(* IEC 61131-3 sources: programs/VI-54/VI-54_20171205/VI-54_20171205/Stations/Screen/LseClass170718/Class/ParameterLogFile, 1 file *)

(* ---- ParameterLogFile.st ---- *)
(*!
<Class
	Name               = "ParameterLogFile"
	Revision           = "0.0"
	RealtimeTask       = "false"
	CyclicTask         = "false"
	BackgroundTask     = "false"
	Sigmatek           = "false"
	OSInterface        = "false"
	HighPriority       = "false"
	Automatic          = "false"
	UpdateMode         = "Prescan"
	SharedCommandTable = "true"
	Objectsize         = "(540,120)">
	<Channels>
	</Channels>
	<Network Name="ParameterLogFile">
		<!-- List of Components in this network -->
		<Components>
			<Object
				Name       = "_base"
				Class      = "_Global"
				Position   = "(218,120)"
				Visualized = "true"
				Remotely   = "true">
				<Channels>
					<Server Name="Server0">
						<OPCSettings WriteProtected="false"/>
					</Server>
					<Client Name="Lse"/>
				</Channels>
			</Object>
		</Components>
		<Comments>
		</Comments>
		<!-- List of Connections in this network -->
		<Connections>
			<Connection Source="this.Server0" Destination="_base.Server0" Vertices="(690,210),(518,210),"/>
			<Connection Source="_base.Lse" Destination="this.Lse" Vertices="(218,210),(38,210),"/>
		</Connections>
		<!-- Headerfiles -->
		<Options>
		</Options>
	</Network>
</Class>
*)
#pragma using _Global

ParameterLogFile : CLASS
: _Global
  //Servers:
  //Clients:
  //Variables:
		VariableInformation 	: ^_EDITOR;
		WindowNbr 	: UDINT;
		ActualValue 	: DINT;
		ActualMin 	: DINT;
		ActualMax 	: DINT;
  //Functions:
				//! <Function Comment="method is called right before the kernel wants to open a toucheditor&#13;&#10;the parameter &apos;pe&apos; is a pointer to structure where the whole editorinformation is shown&#13;&#10;parameter preselect is the windownumber of the editor &#13;&#10;return &apos;preselect&apos; if you want the kernel to open the editor, on the other hand 16#FFFF&#13;&#10;" Name="IF_OpenTouchEditor"/>
	FUNCTION VIRTUAL GLOBAL IF_OpenTouchEditor
		VAR_INPUT
			pe 	: ^_EDITOR;
			preselect 	: UINT;
		END_VAR
		VAR_OUTPUT
			retcode 	: UINT;
		END_VAR;
  //Tables:
	FUNCTION @STD
		VAR_OUTPUT
			ret_code	: CONFSTATES;
		END_VAR;
	FUNCTION GLOBAL TAB @CT_;
END_CLASS;

FUNCTION VIRTUAL GLOBAL ParameterLogFile::IF_OpenTouchEditor
	VAR_INPUT
		pe 	: ^_EDITOR;
		preselect 	: UINT;
	END_VAR
	VAR_OUTPUT
		retcode 	: UINT;
	END_VAR

  WindowNbr := preselect;
  if WindowNbr = 0 then
    VariableInformation := pe;
    ActualValue := VariableInformation^.result.value;
    ActualMin   := VariableInformation^.result.rmin;
    ActualMax   := VariableInformation^.result.rmax;
  end_if;

  retcode := preselect;

END_FUNCTION
